Fanuc KAREL source: ko00081.KL

-- PROVISIONAL review KL for V770-1; original PC SHA256 9cf2623e50d50216f6a560a683a37a71b036037e270893753f61d61bf1908e8e
-- Incomplete behavior may be omitted. Consult companion uncertainty JSON. Do not deploy.
PROGRAM KO00081
%NOLOCKGROUP
BEGIN
  -- UNRESOLVED_PC offsets 5-12; opcodes 9D,23
  -- UNRESOLVED_PC offsets 17-66; opcodes 27,27,49,7E,AD,22,1C,22,31,7E,4A
  -- UNRESOLVED_PC offsets 71-75; opcodes 7F
END KO00081
